Staubli VAL3: page_editTraj.dtx

bool bButton[8]
  [0] = true
  [1] = true
  [2] = true
  [4] = true
  [5] = true
  [6] = true
  [7] = true
bool bExit
bool bLarge
bool bShowStatus
bool bTrigger
num nClockStatus = 962.397
num nIndex
num nIndexItem
num nKey
num nOldIndex
public num nPage
num nRefresh = 1149.353
num nSelected = -1
num nTime = 0.1
num nUserItem = 6
num nView
string sAction[3]
string sEvent = "Name: > appro"
public string sItems = "pick"
string sListUser[6]
  [0] = "appro   X > 0   "
  [1] = "appro   Y > 0   "
  [2] = "appro   Z > -50   "
  [3] = "appro  RX > 0   "
  [4] = "appro  RY > 0   "
  [5] = "appro  RZ > 0   "
string sMenu[8]
  [0] = "Here"
  [1] = "Align"
  [2] = "Tool"
  [4] = "Motion"
  [5] = "Delete"
  [6] = "Insert"
  [7] = "Save"
string sMenu8[8]
string sMenuUser[8]
  [0] = "Here"
  [1] = "Align"
  [2] = "Tool"
string sMessage[2]
  [0] = "ON"
  [1] = "OFF"
string sOldListUser
string sTrajName = "pick"
frame fFather = {fatherId=world[0]}
string sWorkingmode[16]
  [0] = "点属性      >"
  [1] = "Appro X     >"
  [2] = "Appro Y     >"
  [3] = "Appro Z     >"
  [4] = "Appro RX    >"
  [5] = "Appro RY    >"
  [6] = "Appro RZ    >"
  [7] = "速度        >"
  [8] = "加速度      >"
  [9] = "偏移方式    >"
  [10] = "偏移对象    >"
  [11] = "移动方式    >"
  [12] = "停止        >"
  [13] = "混合        >"
  [14] = "信号        >"
  [15] = "提前输出    >"
string sList
num i
public string sTitle
public string sPassword[2]
  [0] = "chenpeng"
  [1] = "xixi"
string sPasswd
